// TIA Portal V20 export
DATA_BLOCK "EmNodes"   // DB3
{ DB_Accessible_From_OPC_UA := 'FALSE' }
AUTHOR : ERsystem_FA2_DH. Kim
// stored: Access Published, DBAccessibleFromOPCUA false, DBAccessibleFromWebserver false, MemoryReserve 100, Namespace Unit1
   VAR
      unitStatus { ExternalWritable := 'False'} : "LAF_typeUnitStatus";   // Status of the unit
      emFeedback { ExternalWritable := 'False'} : Array[0.._.U1_NO_OF_EMs] of "LUC_typeEmFeedback";   // Status of the individual equipment modules
      emRelations : Struct
         em00 : "Unit1.type_emRelations_em0";
         em01 : "Unit1.type_emRelations_em1";
         em02 : "Unit1.type_emRelations_em2";
         em03 : "Unit1.type_emRelations_em3";
         em04 : "Unit1.type_emRelations_em4";
         em05 : "Unit1.type_emRelations_em5";
         em06 : "Unit1.type_emRelations_em6";
         em07 : "Unit1.type_emRelations_em7";
      END_STRUCT;
      emIt { S7_SetPoint := 'True'} : Array[0..13] of "LER_OEM_Data";
      enableControlInterfaces { ExternalWritable := 'False'} : "LAF_typeEnableControlInterfaces";
      oem { ExternalAccessible := 'False'; ExternalVisible := 'False'; ExternalWritable := 'False'; S7_SetPoint := 'True'} : Array[0..10] of "LER_OEM_Data";
      FATModeSelect { ExternalWritable := 'False'} : "LER_TypeFATMode_ModeSelect";
   END_VAR
   VAR RETAIN
      FATModeInterface { ExternalWritable := 'False'} : "LER_TypeFATModeInterface";
   END_VAR
   VAR
      signalStack { ExternalWritable := 'False'} : "LUC_typeSignalStackByBool";
      clock { ExternalWritable := 'False'} : "LAF_typeGlobalClockMem";
      slmRunning { S7_SetPoint := 'True'} : Bool;
      slmPowerOff { ExternalWritable := 'False'} : Bool;
      InterfaceTestMode { ExternalWritable := 'False'} : Bool;
      CapabilityModeComplete { ExternalWritable := 'False'} : Bool;
      SamplingModeComplete { ExternalWritable := 'False'} : Bool;
      stateCommandsExecute { ExternalWritable := 'False'} : Bool;
      atLeastOneDoorUnlock { ExternalWritable := 'False'} : Bool;
      SleepModeActivationTime : Time;
      DeepSleepModeActivationTime : Time;
      SleepModeChangeReq : Bool;
      DeepSleepModeChangeReq : Bool;
      WakeupRecoveryRequired : Bool;
      sleep : Struct
         State { S7_SetPoint := 'True'} : "LER_typeSleepMode";
         command { S7_SetPoint := 'True'} : "LER_typeSleep";
      END_STRUCT;
      "========Communication========" { ExternalWritable := 'False'} : Bool;
      BA010 { ExternalWritable := 'False'} : "LER_typeCommunicationReelCut";
      BA015 { ExternalWritable := 'False'} : "LER_typeCommunicationReelCut";
      BA030 { ExternalWritable := 'False'} : "LER_typeCommunicationStack";
      BA060 { S7_SetPoint := 'True'} : "LER_typeCommunicationInspection";
      "========Safety========" { ExternalWritable := 'False'} : Bool;
      devicesSummary : "LWONIK_typeDevicesStatusSummary";
      safetyZone1OpEnable { ExternalWritable := 'False'} : "LWONIK_typeSafetyZoneManualOperation";
      safetyZone2OpEnable { ExternalWritable := 'False'} : "LWONIK_typeSafetyZoneManualOperation";
      safetyZone3OpEnable { ExternalWritable := 'False'} : "LWONIK_typeSafetyZoneManualOperation";
      doorOpenRequest : Bool;
      safetyStatusZone1 { S7_SetPoint := 'True'} : "LWONIK_typeZoneStatus";
      safetyStatusZone2 { S7_SetPoint := 'True'} : "LWONIK_typeZoneStatus";
      safetyStatusZone3 { S7_SetPoint := 'True'} : "LWONIK_typeZoneStatus";
      mainOpMode : "LWONIK_typeOperationMode";
      pHmiMode { ExternalWritable := 'False'} : "LWONIK_typePhmiMode";
      scsMode { ExternalWritable := 'False'} : "LWONIK_typeScsMode";
      rcMode1 { S7_SetPoint := 'True'} : "LWONIK_typeRollChangeMode";
      rcMode2 { S7_SetPoint := 'True'} : "LWONIK_typeRollChangeMode";
      scrapBox1 { S7_SetPoint := 'True'} : "LWONIK_typeScrapBox";
      scrapBox2 { S7_SetPoint := 'True'} : "LWONIK_typeScrapBox";
      SafetySensor { S7_SetPoint := 'True'} : "LWONIK_typeSafetySensor";
      EstopStatus { ExternalWritable := 'False'} : "LWONIK_typeFromSafetyEstopStatus";
      FdoorStatus { ExternalWritable := 'False'} : "LWONIK_typeFromSafetyDoorStatus";
      fDoorDrive { S7_SetPoint := 'True'} : "Safety.typeFDoorFunction";
      cvConverStatus : Struct
         cvCoverOK1 : Bool;
         cvCoverOK2 : Bool;
         cvCoverAllOK : Bool;
         cvCoverSystemFaults : Bool;
      END_STRUCT;
      AllSFDoorOpen { S7_SetPoint := 'True'} : Bool;
      AllFDoorClosed : Bool;
      OpHmiOperationEnable : Bool;
      PHmiOperationEnable : Bool;
      FullStepReady : Bool;
      MobilePanelConnected : Bool;
      MobilePanelPermissions : Bool;
      SS1TimeExtension : Bool;
      EnableServoAck : Bool;
      BA10SCSModeSelect : Bool;
      BA15SCSModeSelect : Bool;
      BA30SCSModeSelect : Bool;
      BA60SCSModeSelect : Bool;
      "=======ETC========" : Bool;
      allBrakeTest { ExternalWritable := 'False'} : "LER_typeBrakeTestUnitInterface";
      booltest { S7_SetPoint := 'True'} : Array[0..15] of Bool;
      motionInterface : Struct
         Dancer : Struct
            Enable : Bool := FALSE;
            Stop : Bool := FALSE;
            Reset : Bool := FALSE;
         END_STRUCT;
         StackMain : Struct
            Calculate : Bool := FALSE;
            SemiStep : Bool := FALSE;
            FullStep : Bool := FALSE;
            AutoReady : Bool := FALSE;
            AutoStart : Bool := FALSE;
            StopMotion : Bool := FALSE;
            StopForCalculate : Bool;
            Reset : Bool := FALSE;
         END_STRUCT;
      END_STRUCT;
      FullStepRun : Bool;
      MotionRunlockBit : Bool;   // Motion Busy
      MotionReady : Bool;
      BA60ExternalDoorOpen : Bool;
   END_VAR
BEGIN
   // emRelations.em06.sequence.Spare1.preOperationCheck.Bool1 : FinalRoller In CathodePos
   // emRelations.em06.sequence.Spare1.preOperationCheck.Bool2 : FinalRoller In AnodePos
   // emRelations.em07."Bool"[1] : SepaGripperAxisX Move To BA60
   // BA010.ReelCutToStack.UnitStatus.specialFunctions.specialFunction1 : gaugeR&rType1
   // BA010.ReelCutToStack.UnitStatus.specialFunctions.specialFunction2 : gaugeR&rType3
   // BA010.ReelCutToStack.UnitStatus.specialFunctions.specialFunction3 : releaseEntry
   // BA010.ReelCutToStack.UnitStatus.specialFunctions.specialFunction4 : dryRun
   // BA010.ReelCutToStack.UnitStatus.specialFunctions.specialFunction5 : runOut
   // BA010.ReelCutToStack.UnitStatus.specialFunctions.specialFunction6 : reWrokMode
   // BA010.ReelCutToStack.UnitStatus.specialFunctions.specialFunction7 : specialFunction7
   // BA010.ReelCutToStack.UnitStatus.specialFunctions.specialFunction8 : specialFunction8
   // BA010.ReelCutToStack.UnitStatus.specialFunctions.specialFunction9 : visionUnuse
   // BA010.ReelCutToStack.UnitStatus.specialFunctions.specialFunction10 : qrReadVisionPosUnuse
   // BA010.ReelCutToStack.UnitStatus.specialFunctions.specialFunction11 : qrReadStk1PosUnuse
   // BA010.ReelCutToStack.UnitStatus.specialFunctions.specialFunction12 : qrReadStk2PosUnuse
   // BA010.ReelCutToStack.UnitStatus.specialFunctions.specialFunction13 : identRFIDReadUnuse
   // BA010.ReelCutToStack.UnitStatus.specialFunctions.specialFunction14 : specialFunction14
   // BA010.ReelCutToStack.UnitStatus.specialFunctions.specialFunction15 : stack1InterfaceUnuse
   // BA010.ReelCutToStack.UnitStatus.specialFunctions.specialFunction16 : stack2InterfaceUnuse
   // BA010.ReelCutToStack.InterfaceData."Bool"[0] : Load Enable
   // BA010.ReelCutToStack.InterfaceData."Bool"[1] : Load Complete Comfirm
   // BA010.ReelCutToStack.InterfaceData."Bool"[2] : Cell Data Report
   // BA010.ReelCutToStack.InterfaceData."Bool"[10] : Motion Auto Ready
   // BA010.ReelCutToStack.InterfaceData."Bool"[11] : Motion Auto Start
   // BA010.ReelCutToStack.InterfaceData."Bool"[12] : Motion Auto Stop
   // BA010.StackToReelCut.InterfaceData."Bool"[0] : Load Requset
   // BA010.StackToReelCut.InterfaceData."Bool"[1] : Load Busy
   // BA010.StackToReelCut.InterfaceData."Bool"[2] : Load Complete
   // BA010.StackToReelCut.InterfaceData."Bool"[3] : Cell Data Request
   // BA010.StackToReelCut.InterfaceData."Bool"[4] : Cell Data Report Ack
   // BA010.StackToReelCut.InterfaceData."Bool"[5] : Cell Data Report Nck
   // BA010.StackToReelCut.InterfaceData."Bool"[10] : Motion Auto Ready
   // BA010.StackToReelCut.InterfaceData."Bool"[11] : Motion Auto Start
   // BA010.StackToReelCut.InterfaceData."Bool"[12] : Motion Auto Stop
   // BA015.ReelCutToStack.InterfaceData."Bool"[0] : Load Enable
   // BA015.ReelCutToStack.InterfaceData."Bool"[1] : Load Complete Comfirm
   // BA015.ReelCutToStack.InterfaceData."Bool"[2] : Cell Data Report
   // BA015.ReelCutToStack.InterfaceData."Bool"[10] : Motion Auto Ready
   // BA015.ReelCutToStack.InterfaceData."Bool"[11] : Motion Auto Start
   // BA015.ReelCutToStack.InterfaceData."Bool"[12] : Motion Auto Stop
   // BA015.StackToReelCut.InterfaceData."Bool"[0] : Load Requset
   // BA015.StackToReelCut.InterfaceData."Bool"[1] : Load Busy
   // BA015.StackToReelCut.InterfaceData."Bool"[2] : Load Complete
   // BA015.StackToReelCut.InterfaceData."Bool"[3] : Cell Data Request
   // BA015.StackToReelCut.InterfaceData."Bool"[4] : Cell Data Report Ack
   // BA015.StackToReelCut.InterfaceData."Bool"[5] : Cell Data Report Nck
   // BA015.StackToReelCut.InterfaceData."Bool"[10] : Motion Auto Ready
   // BA015.StackToReelCut.InterfaceData."Bool"[11] : Motion Auto Start
   // BA015.StackToReelCut.InterfaceData."Bool"[12] : Motion Auto Stop
   // BA060.InspectionToStack.InterfaceData."Bool"[0] : Heartbeat
   // BA060.InspectionToStack.InterfaceData."Bool"[1] : ReadyForOperation
   // BA060.InspectionToStack.InterfaceData."Bool"[2] : ReachedHome
   // BA060.InspectionToStack.InterfaceData."Bool"[3] : MachineInOperation
   // BA060.InspectionToStack.InterfaceData."Bool"[4] : LoaderOutsideModule
   // BA060.InspectionToStack.InterfaceData."Bool"[5] : LoaderOutsideCollision
   // BA060.InspectionToStack.InterfaceData."Bool"[10] : PartClamped
   // BA060.InspectionToStack.InterfaceData."Bool"[11] : PartUnclamped
   // BA060.InspectionToStack.InterfaceData."Bool"[16] : RequestUnclamp
   // BA060.InspectionToStack.InterfaceData."Bool"[17] : PartOn
   // BA060.InspectionToStack.InterfaceData."Bool"[18] : RequestPart
   // BA060.InspectionToStack.InterfaceData."Bool"[19] : OnPositionUnloading
   // BA060.InspectionToStack.InterfaceData."Bool"[22] : RequestCollisionON
   // BA060.InspectionToStack.InterfaceData."Bool"[23] : UnoadComplete
   // BA060.InspectionToStack.InterfaceData."Bool"[26] : DataCatchUp
   // BA060.InspectionToStack.InterfaceData."Bool"[27] : DataCompareOK
   // BA060.InspectionToStack.InterfaceData."Bool"[28] : DataDeleted
   // BA060.InspectionToStack.InterfaceData."Bool"[32] : NG RequestPart
   // BA060.InspectionToStack.InterfaceData."Bool"[33] : NG RequestUnclamp
   // BA060.InspectionToStack.InterfaceData."Bool"[34] : NG UnoadComplete
   // BA060.InspectionToStack.InterfaceData."Bool"[48] : ReturnToHome
   // BA060.InspectionToStack.InterfaceData."Bool"[49] : AutoStart
   // BA060.InspectionToStack.InterfaceData."Bool"[50] : EndOfCycle
   // BA060.InspectionToStack.InterfaceData."Bool"[51] : RequestGateOpen
   // BA060.StackToInspection.InterfaceData."Bool"[0] : Heartbeat
   // BA060.StackToInspection.InterfaceData."Bool"[1] : ReadyForOperation
   // BA060.StackToInspection.InterfaceData."Bool"[2] : ReachedHome
   // BA060.StackToInspection.InterfaceData."Bool"[3] : MachineInOperation
   // BA060.StackToInspection.InterfaceData."Bool"[4] : NoInterference
   // BA060.StackToInspection.InterfaceData."Bool"[10] : PartClamped
   // BA060.StackToInspection.InterfaceData."Bool"[11] : PartUnclamped
   // BA060.StackToInspection.InterfaceData."Bool"[16] : RequestClamp
   // BA060.StackToInspection.InterfaceData."Bool"[17] : PartOn
   // BA060.StackToInspection.InterfaceData."Bool"[18] : PartReady
   // BA060.StackToInspection.InterfaceData."Bool"[19] : LoaderInTranferArea
   // BA060.StackToInspection.InterfaceData."Bool"[20] : CollisionAreaOn
   // BA060.StackToInspection.InterfaceData."Bool"[21] : CollisionAreaOff
   // BA060.StackToInspection.InterfaceData."Bool"[23] : LoadComplete
   // BA060.StackToInspection.InterfaceData."Bool"[26] : DataCatchUp
   // BA060.StackToInspection.InterfaceData."Bool"[27] : DataCompareOK
   // BA060.StackToInspection.InterfaceData."Bool"[28] : DataDeleted
   // BA060.StackToInspection.InterfaceData."Bool"[32] : NG PartReady
   // BA060.StackToInspection.InterfaceData."Bool"[33] : NG RequestClamp
   // BA060.StackToInspection.InterfaceData."Bool"[34] : NG LoadComplete
   // BA060.StackToInspection.InterfaceData."Bool"[48] : ReturnToHome
   // BA060.StackToInspection.InterfaceData."Bool"[49] : AutoStart
   // BA060.StackToInspection.InterfaceData."Bool"[50] : EndOfCycle
   // BA060.StackToInspection.InterfaceData."Bool"[51] : StopForOpenGate
   booltest[0] := True;
END_DATA_BLOCK
